FUNCTION_BLOCK EL3001
VAR
	_io : EL3xx1_Data;
	{attribute addProperty Name "WcState"}
	_wcState : WcStateInputToggle;
	{attribute addProperty Name "Info data"}
	_infoData : InfoDataAds;
END_VAR

PROPERTY IO : REFERENCE TO EL3xx1_Data
GET
IO REF= _io;
END_GET
END_PROPERTY

PROPERTY WcState : REFERENCE TO WcStateInputToggle
GET
WcState REF= _wcState;
END_GET
END_PROPERTY

END_FUNCTION_BLOCK

(* stored: Version 1.1.0.1, ProductVersion 3.1.4024.9
   POU EL3001: Id {00ca6e78-ad1d-0c27-3710-d424f43db701}, SpecialFunc None
   Property IO: Id {842e7815-184d-01e6-2fe6-6f39e76935dd}
   Get Get: Id {3e24745a-b35c-03f2-2e00-54d3bd5a64dd}
   Property WcState: Id {88fd9bca-c6d8-0de4-2aee-5ead4f3337ee}
   Get Get: Id {7a0e0394-be28-0593-0330-e20111d92340} *)
